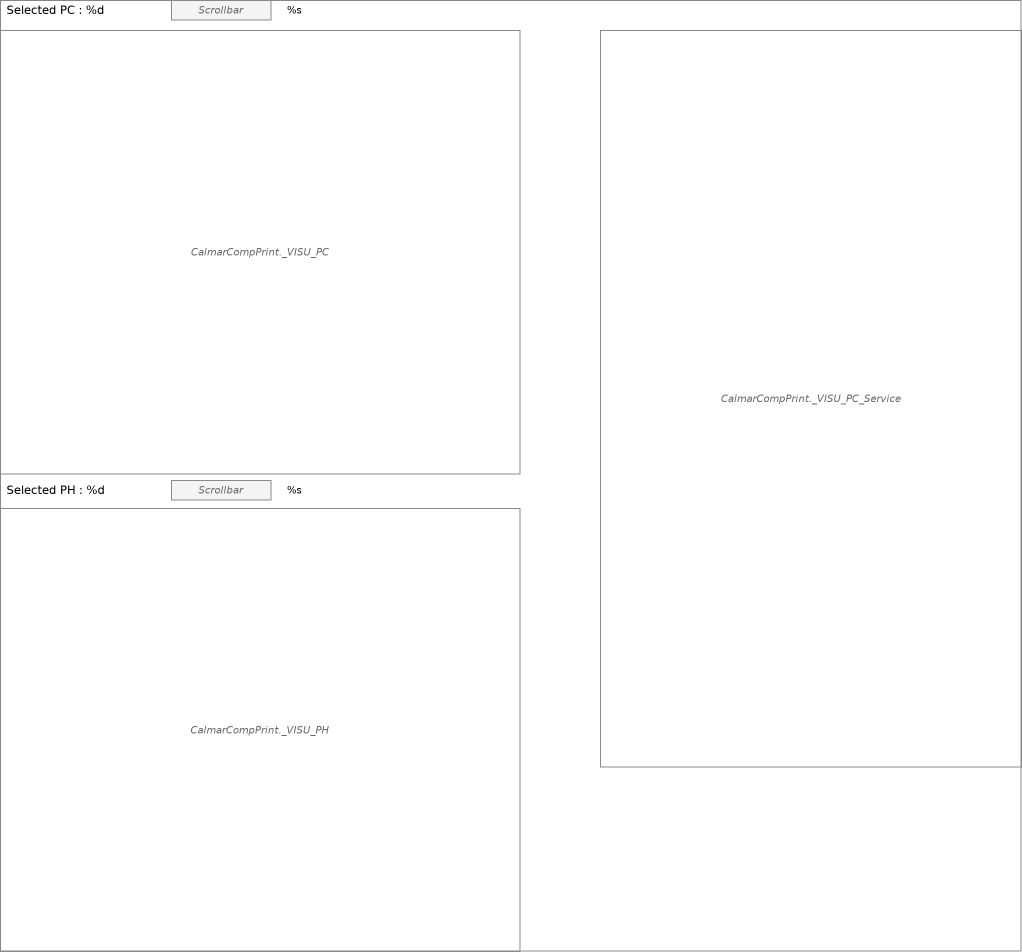
VISUALIZATION _VISU_Hardware  // 1022x952
VAR_IN_OUT
	  m_fbHw  : FB_HardwarePool;      (*visu fb instance*)
END_VAR
    Frame (600,30 422x737)
        shows CalmarCompPrint._VISU_PC_Service(m_Inst := m_fbHw._rPcVisuSel^)
    Rectangle (0,0 157x20), "Selected PC : %d", text variable: m_fbHw.fBPcSelector.pSelect^
        OnMouseDown: write the text variable via Edit, min m_fbHw.fBPcSelector.iBoundLower, max m_fbHw.fBPcSelector.iBoundUpper
    Scrollbar (171,0 100x20)
        p3598130195: m_fbHw.fBPcSelector.iBoundLower
        p2245068023: m_fbHw.fBPcSelector.iBoundUpper
        p1057716461: m_fbHw.fBPcSelector.pSelect^
    Rectangle (284,0 248x20), "%s", text variable: m_fbHw._rAdsPcVisuSel^.aO_Name
    Frame (0,30 520x444)
        shows CalmarCompPrint._VISU_PC(m_Inst := m_fbHw._rPcVisuSel^)
    Rectangle (0,480 157x20), "Selected PH : %d", text variable: m_fbHw.fBPhSelector.pSelect^
        OnMouseDown: write the text variable via Edit, min m_fbHw.fBPhSelector.iBoundLower, max m_fbHw.fBPhSelector.iBoundUpper
    Scrollbar (171,480 100x20)
        p3598130195: m_fbHw.fBPhSelector.iBoundLower
        p2245068023: m_fbHw.fBPhSelector.iBoundUpper
        p1057716461: m_fbHw.fBPhSelector.pSelect^
    Rectangle (284,480 248x20), "%s", text variable: m_fbHw._rAdsPhVisuSel^.aO_Name
    Frame (0,508 520x444)
        shows CalmarCompPrint._VISU_PH(m_Inst := m_fbHw._rPhVisuSel^)
END_VISUALIZATION

(* stored: Version 1.1.0.1, ProductVersion 3.1.4024.11
   Visu _VISU_Hardware: Id {b94d3190-9292-476b-a4e2-24c388bd60d9} *)
